FUNCTION_BLOCK AR2_REAL_TO_R (* Composite FB for convert REAL to AR2 *)
  (* Standard: 61499-2; Description: Copyright (c) 2024 HR Agrartechnik GmbH This program and the accompanying materials are made available under the terms of the Eclipse Public License 2.0 which is available at https://www.eclipse.org/legal/epl-2.0/ SPDX-License-Identifier: EPL-2.0 *)
  (* Version 1.0, 2024-04-24, Franz Höpfinger, HR Agrartechnik GmbH *)
  PACKAGE adapter::conversion::bidirectional;
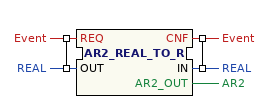
  EVENT_INPUT
    REQ WITH OUT; (* Request to Adapter *)
  END_EVENT
  EVENT_OUTPUT
    CNF WITH IN; (* Confirmation from Adapter *)
  END_EVENT
  VAR_INPUT
    OUT : REAL;
  END_VAR
  VAR_OUTPUT
    IN : REAL; (* Input data from Adapter *)
  END_VAR
  PLUGS
    AR2_OUT : adapter::types::bidirectional::AR2; (* Adapter Output *)
  END_PLUGS
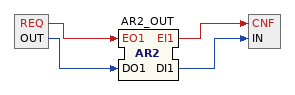
  EVENT_CONNECTIONS
    REQ TO AR2_OUT.EO1;
    AR2_OUT.EI1 TO CNF;
  END_CONNECTIONS
  DATA_CONNECTIONS
    OUT TO AR2_OUT.DO1;
    AR2_OUT.DI1 TO IN;
  END_CONNECTIONS
END_FUNCTION_BLOCK
